(* Logix 5000 project; controller DC01 vendor 1 type 14 code 165 rev 32.12; software revision 32.04; part 3 of 13 *)
(* tags used below, declared in another part *)
   Break_1stStation : BOOL;
   Break_LineWide : BOOL;
   Break_WorkCenter : BOOL;
   Break_Workstation : BOOL;
   FaultExists : CONTROL;
   LN01_MainLine_MSG : MESSAGE;
   Local_Timer : TIMER[30];
   local_timer2 : TIMER;
   ONS_0 : DINT;
   Shift_Reset_ONS : BOOL;
   Barcode_Scan : MESSAGE;
   LN01_1st_Station_Break_Code : DINT;
   LN01_Boxing_MNT : DINT;
   LN01_Ceran_MNT : DINT;
   LN01_Console_MNT : DINT;
   LN01_Cooktop_MNT : DINT;
   LN01_Current_Shift_Duration_Mins : DINT;
   LN01_Current_Shift_Duration_wBreaks_Mins : DINT;
   LN01_DC_Controlled_Theoretical_Units : BOOL;
   LN01_Door_MNT : DINT;
   LN01_FPY : DINT;
   LN01_FrontFrame_MNT : DINT;
   LN01_Ignition_NewSNModel : BOOL[32];
   LN01_Ignition_SNModelMSG : STRING[5];
   LN01_MachineOverAll_MNT : DINT;
   LN01_Main_Messages : DINT[250];
   LN01_MainBack_MNT : DINT;
   LN01_Messages_Barcode_SNModel : Barcode_SNModel;
   LN01_OvenCavity_MNT : DINT;
   LN01_Schedule : UDT_Current_Status;
   LN01_Schedule_Cycle_Timer : TIMER;
   LN01_Schedule_Max_Break_Duration : DINT;
   LN01_Schedule_Max_Break_Timer : TIMER;
   LN01_Schedule_TAKT : REAL;
   LN01_Scheduled_Units_Buffer : DINT;
   LN01_SidePanels_MNT : DINT;
   LN01_StorageDrawer_MNT : DINT;
   LN01_Test_MNT : DINT;
   LN01_Theoretical_Units_Counter : COUNTER;
   LN01_Theoretical_Units_Counter_ONS : BOOL;
   LN01_Units_for_repair : DINT;
   LN01_Wiring_MNT : DINT;
   LN01ECM02 : DINT;
   LN01ECM03 : DINT;
   LN01ECM04 : DINT;
   LN01ECM05 : DINT;
   LN01EDM04 : DINT;
   LN01EDM06 : DINT;
   LN01EDM07 : DINT;
   LN01EDM08 : DINT;
   LN01EEM01 : DINT;
   LN01EEM02 : DINT;
   LN01EEM03 : DINT;
   LN01EES01 : DINT;
   LN01EES02 : DINT;
   LN01EES03 : DINT;
   LN01EES04 : DINT;
   LN01EFS04 : DINT;
   LN01EFS05 : DINT;
   LN01EGM04 : DINT;
   LN01EHM01 : DINT;
   LN01EHM02 : DINT;
   LN01EHM03 : DINT;
   LN01EHM04 : DINT;
   LN01EHM05 : DINT;
   LN01EHM06 : DINT;
   LN01EHM07 : DINT;
   LN01EHM08 : DINT;
   LN01NAS01 : DINT;
   LN01NAS02 : DINT;
   LN01NAS03 : DINT;
   LN01NBS02 : DINT;
   LN01SAS03 : DINT;
   LN01SBS01 : DINT;
   LN01SBS03 : DINT;
   LN01SFS03 : DINT;
   LN01WAM01 : DINT;
   LN01WBM01 : DINT;
   LN01WBM02 : DINT;
   LN01WBM03 : DINT;
   LN01WBM04 : DINT;
   LN01WCM01 : DINT;
   LN01WCM02 : DINT;
   LN01WCM03 : DINT;
   LN01WCM04 : DINT;
   LN01WCM05 : DINT;
   LN01WCM06 : DINT;
   LN01WDM01 : DINT;
   LN01WDM02 : DINT;
   LN01WDM03 : DINT;
   LN01WDM04 : DINT;
   LN01WDM05 : DINT;
   LN01WFS01 : DINT;
   LN01WFS02 : DINT;
   LN01WGM01 : DINT;
   LN01WGM02 : DINT;
   LN01WGM03 : DINT;
   LN01WGM04 : DINT;
   LN01WGM05 : DINT;
   LN01WHM08 : DINT;
(* LN01, continued *)

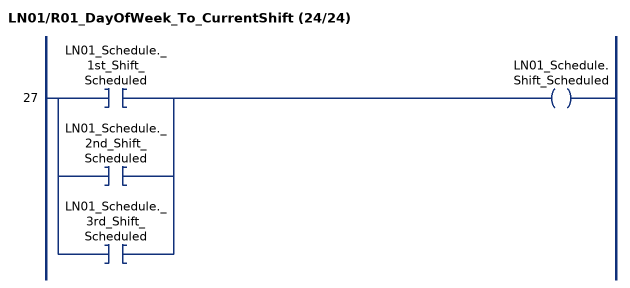
   [picture p24: LN01/R01_DayOfWeek_To_CurrentShift rungs 27-27]
   27: [XIC(LN01_Schedule._1st_Shift_Scheduled) ,XIC(LN01_Schedule._2nd_Shift_Scheduled) ,XIC(LN01_Schedule._3rd_Shift_Scheduled) ]OTE(LN01_Schedule.Shift_Scheduled);
END_ROUTINE

ROUTINE R02_CurrentShift_Calcs   (* ladder *)
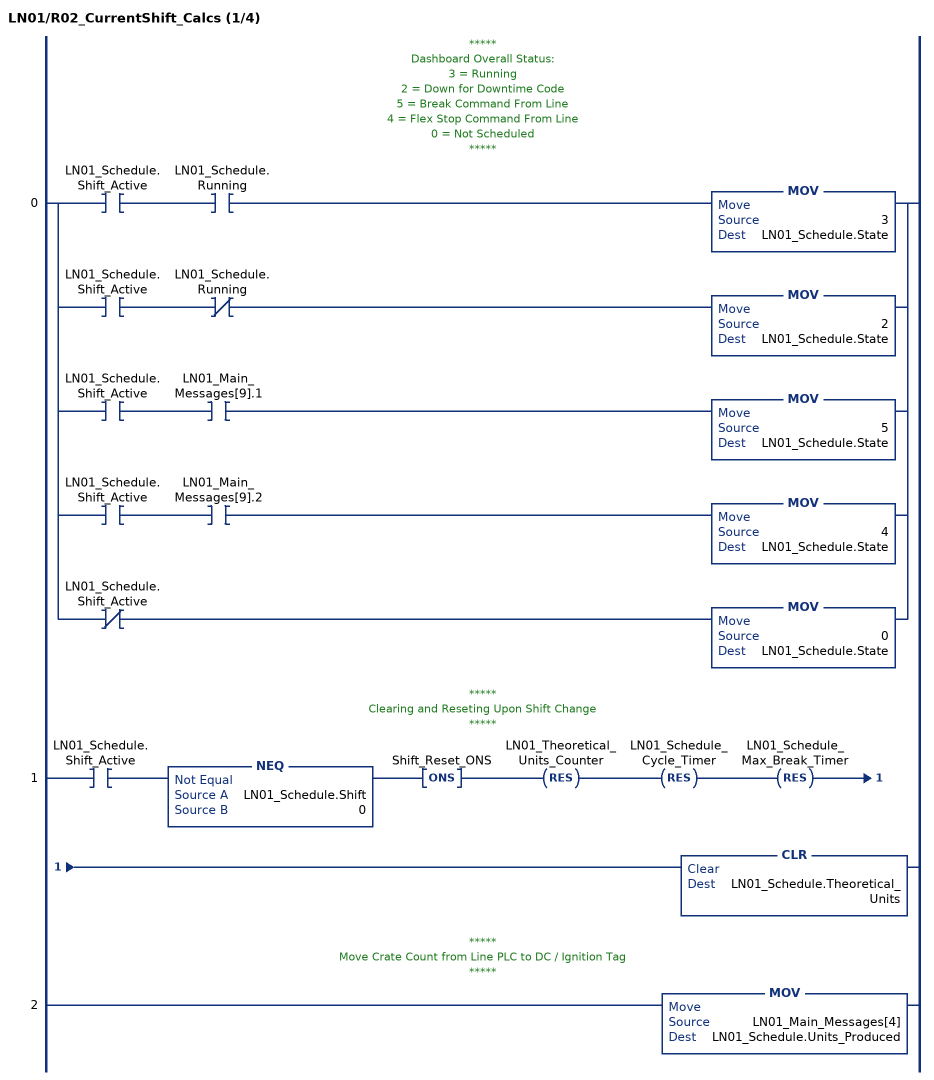
   // *****
   // Dashboard Overall Status:
   // 3 = Running
   // 2 = Down for Downtime Code
   // 5 = Break Command From Line
   // 4 = Flex Stop Command From Line
   // 0 = Not Scheduled
   // *****
   0: [XIC(LN01_Schedule.Shift_Active) XIC(LN01_Schedule.Running) MOV(3,LN01_Schedule.State) ,XIC(LN01_Schedule.Shift_Active) XIO(LN01_Schedule.Running) MOV(2,LN01_Schedule.State) ,XIC(LN01_Schedule.Shift_Active) XIC(LN01_Main_Messages[9].1) MOV(5,LN01_Schedule.State) ,XIC(LN01_Schedule.Shift_Active) XIC(LN01_Main_Messages[9].2) MOV(4,LN01_Schedule.State) ,XIO(LN01_Schedule.Shift_Active) MOV(0,LN01_Schedule.State) ];
   // *****
   // Clearing and Reseting Upon Shift Change
   // *****
   1: XIC(LN01_Schedule.Shift_Active)NEQ(LN01_Schedule.Shift,0)ONS(Shift_Reset_ONS)RES(LN01_Theoretical_Units_Counter)RES(LN01_Schedule_Cycle_Timer)RES(LN01_Schedule_Max_Break_Timer)CLR(LN01_Schedule.Theoretical_Units);
   // *****
   // Move Crate Count from Line PLC to DC / Ignition Tag
   // *****
   2: MOV(LN01_Main_Messages[4],LN01_Schedule.Units_Produced);
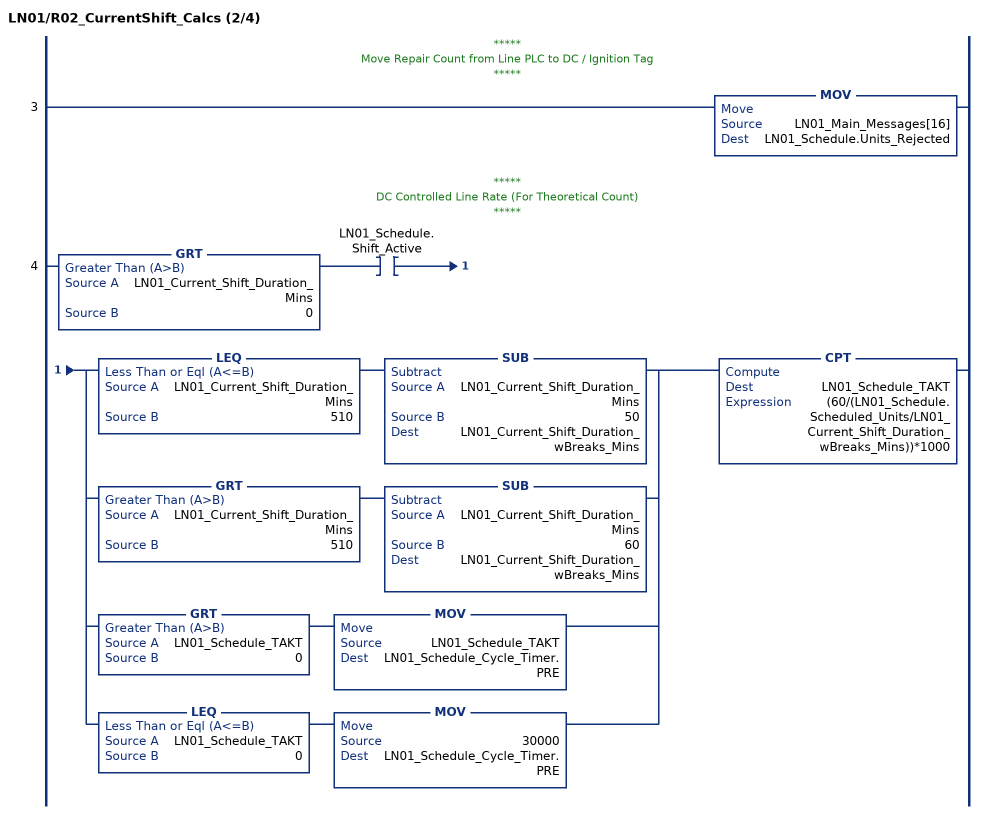
   // *****
   // Move Repair Count from Line PLC to DC / Ignition Tag
   // *****
   3: MOV(LN01_Main_Messages[16],LN01_Schedule.Units_Rejected);
   // *****
   // DC Controlled Line Rate (For Theoretical Count)
   // *****
   4: GRT(LN01_Current_Shift_Duration_Mins,0)XIC(LN01_Schedule.Shift_Active)[LEQ(LN01_Current_Shift_Duration_Mins,510) SUB(LN01_Current_Shift_Duration_Mins,50,LN01_Current_Shift_Duration_wBreaks_Mins) ,GRT(LN01_Current_Shift_Duration_Mins,510) SUB(LN01_Current_Shift_Duration_Mins,60,LN01_Current_Shift_Duration_wBreaks_Mins) ,GRT(LN01_Schedule_TAKT,0) MOV(LN01_Schedule_TAKT,LN01_Schedule_Cycle_Timer.PRE) ,LEQ(LN01_Schedule_TAKT,0) MOV(30000,LN01_Schedule_Cycle_Timer.PRE) ]CPT(LN01_Schedule_TAKT,(60/(LN01_Schedule.Scheduled_Units/LN01_Current_Shift_Duration_wBreaks_Mins))*1000);
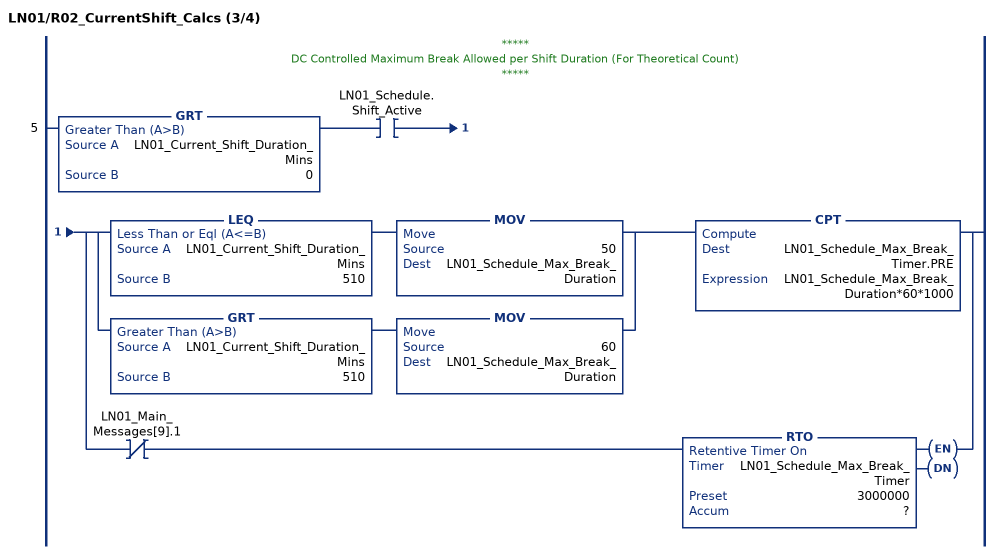
   // *****
   // DC Controlled Maximum Break Allowed per Shift Duration (For Theoretical Count)
   // *****
   5: GRT(LN01_Current_Shift_Duration_Mins,0)XIC(LN01_Schedule.Shift_Active)[[LEQ(LN01_Current_Shift_Duration_Mins,510) MOV(50,LN01_Schedule_Max_Break_Duration) ,GRT(LN01_Current_Shift_Duration_Mins,510) MOV(60,LN01_Schedule_Max_Break_Duration) ] CPT(LN01_Schedule_Max_Break_Timer.PRE,LN01_Schedule_Max_Break_Duration*60*1000) ,XIO(LN01_Main_Messages[9].1) RTO(LN01_Schedule_Max_Break_Timer,?,?) ];
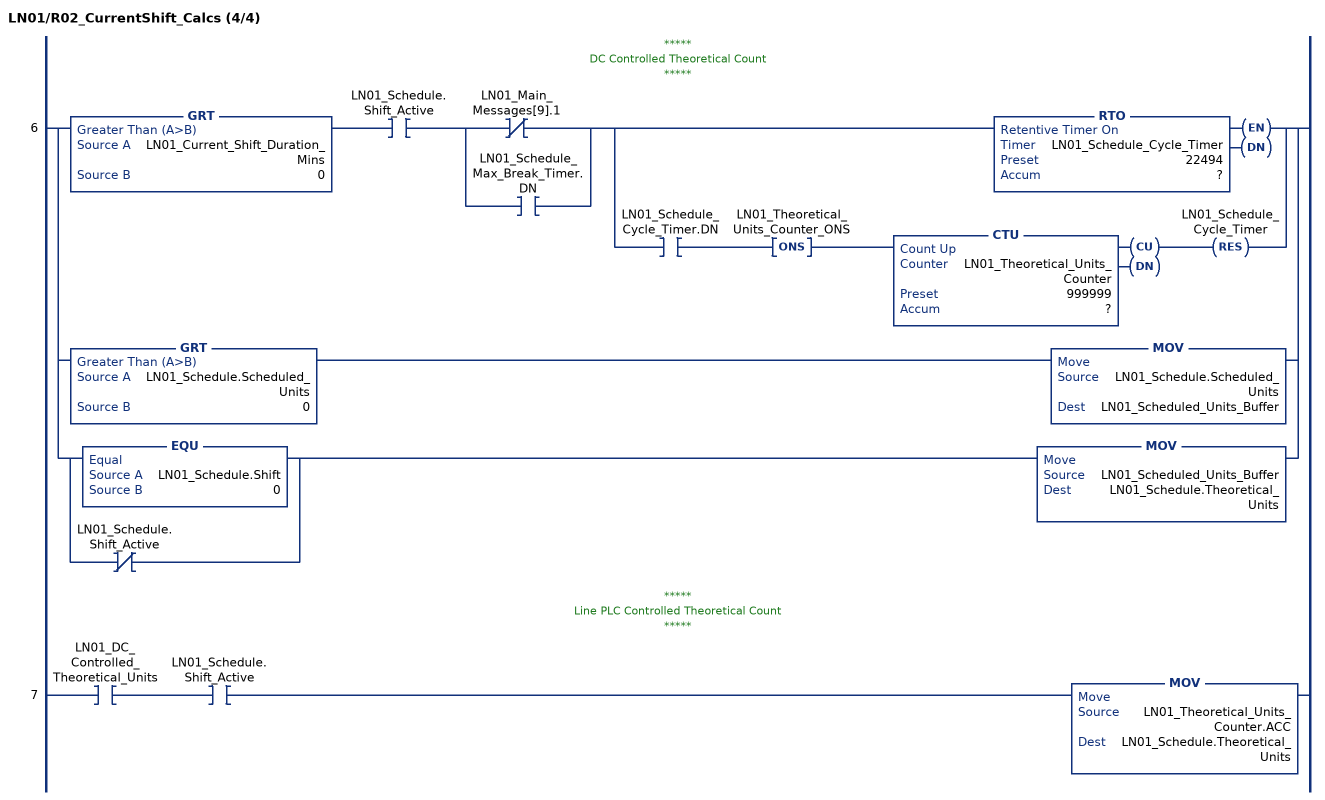
   // *****
   // DC Controlled Theoretical Count
   // *****
   6: [GRT(LN01_Current_Shift_Duration_Mins,0) XIC(LN01_Schedule.Shift_Active) [XIO(LN01_Main_Messages[9].1) ,XIC(LN01_Schedule_Max_Break_Timer.DN) ] [RTO(LN01_Schedule_Cycle_Timer,?,?) ,XIC(LN01_Schedule_Cycle_Timer.DN) ONS(LN01_Theoretical_Units_Counter_ONS) CTU(LN01_Theoretical_Units_Counter,?,?) RES(LN01_Schedule_Cycle_Timer) ] ,GRT(LN01_Schedule.Scheduled_Units,0) MOV(LN01_Schedule.Scheduled_Units,LN01_Scheduled_Units_Buffer) ,[EQU(LN01_Schedule.Shift,0) ,XIO(LN01_Schedule.Shift_Active) ] MOV(LN01_Scheduled_Units_Buffer,LN01_Schedule.Theoretical_Units) ];
   // *****
   // Line PLC Controlled Theoretical Count
   // *****
   7: XIC(LN01_DC_Controlled_Theoretical_Units)XIC(LN01_Schedule.Shift_Active)MOV(LN01_Theoretical_Units_Counter.ACC,LN01_Schedule.Theoretical_Units);
END_ROUTINE

ROUTINE R03_DataFromLines   (* ladder *)
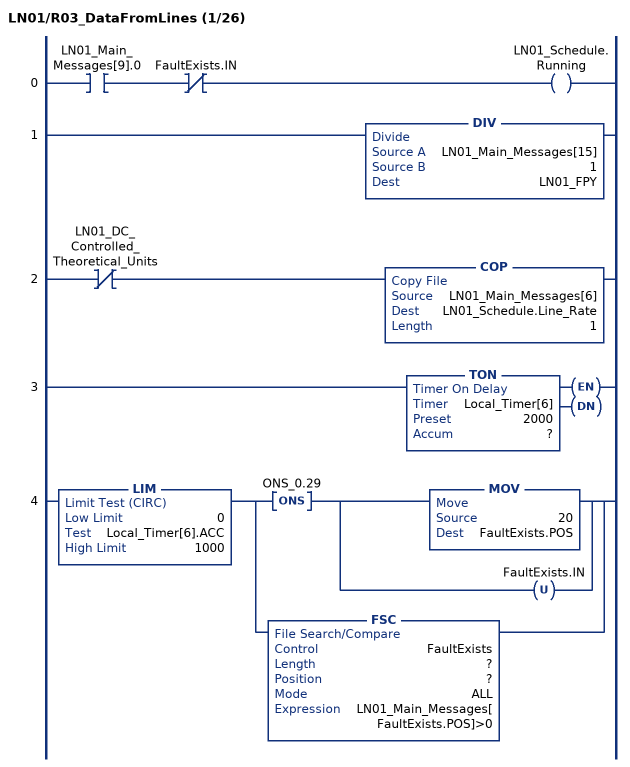
   0: XIC(LN01_Main_Messages[9].0)XIO(FaultExists.IN)OTE(LN01_Schedule.Running);
   1: DIV(LN01_Main_Messages[15],1,LN01_FPY);
   2: XIO(LN01_DC_Controlled_Theoretical_Units)COP(LN01_Main_Messages[6],LN01_Schedule.Line_Rate,1);
   3: TON(Local_Timer[6],?,?);
   4: LIM(0,Local_Timer[6].ACC,1000)[ONS(ONS_0.29) [MOV(20,FaultExists.POS) ,OTU(FaultExists.IN) ] ,FSC(FaultExists,?,?,ALL,LN01_Main_Messages[FaultExists.POS]>0) ];
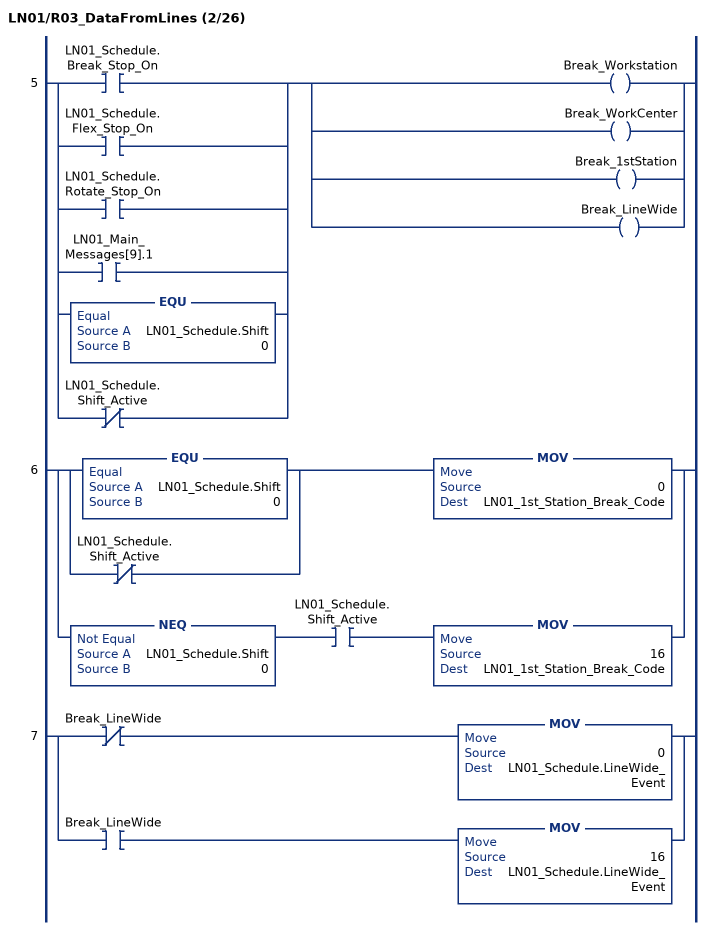
   5: [XIC(LN01_Schedule.Break_Stop_On) ,XIC(LN01_Schedule.Flex_Stop_On) ,XIC(LN01_Schedule.Rotate_Stop_On) ,XIC(LN01_Main_Messages[9].1) ,EQU(LN01_Schedule.Shift,0) ,XIO(LN01_Schedule.Shift_Active) ][OTE(Break_Workstation) ,OTE(Break_WorkCenter) ,OTE(Break_1stStation) ,OTE(Break_LineWide) ];
   6: [[EQU(LN01_Schedule.Shift,0) ,XIO(LN01_Schedule.Shift_Active) ] MOV(0,LN01_1st_Station_Break_Code) ,NEQ(LN01_Schedule.Shift,0) XIC(LN01_Schedule.Shift_Active) MOV(16,LN01_1st_Station_Break_Code) ];
   7: [XIO(Break_LineWide) MOV(0,LN01_Schedule.LineWide_Event) ,XIC(Break_LineWide) MOV(16,LN01_Schedule.LineWide_Event) ];
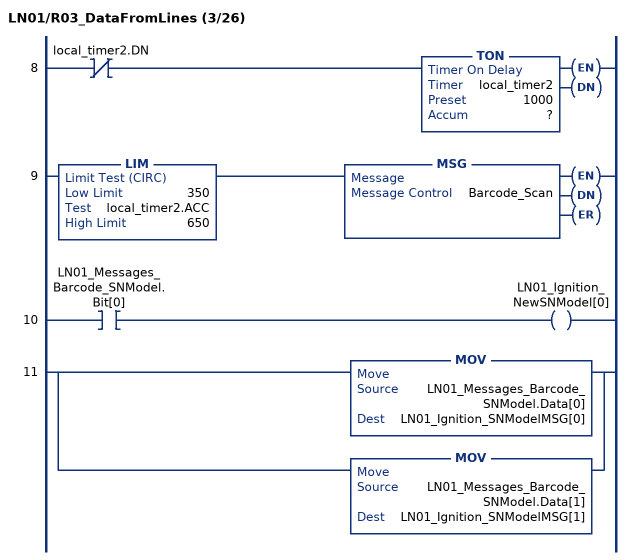
   8: XIO(local_timer2.DN)TON(local_timer2,?,?);
   9: LIM(350,local_timer2.ACC,650)MSG(Barcode_Scan);
   10: XIC(LN01_Messages_Barcode_SNModel.Bit[0])OTE(LN01_Ignition_NewSNModel[0]);
   11: [MOV(LN01_Messages_Barcode_SNModel.Data[0],LN01_Ignition_SNModelMSG[0]) ,MOV(LN01_Messages_Barcode_SNModel.Data[1],LN01_Ignition_SNModelMSG[1]) ];
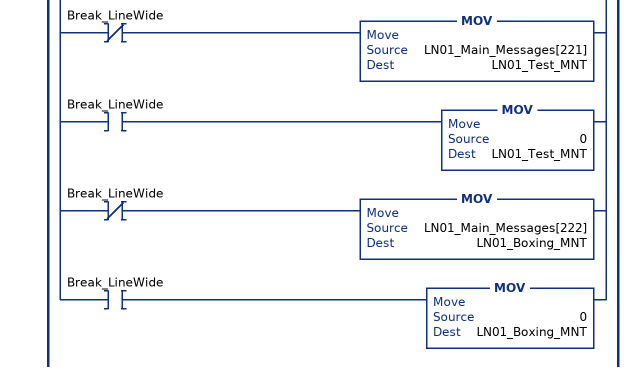
   // MNT Faults
   // If an MNT workcenter is tied to the main line or subline where there is already a workcenter with a workstaiton where "Break_LineWide (when high) MOVEs a 16 in, then that MNT can MOVE a 0 in when "Break_LineWide" goes high
   // If it is an independent MNT (not tied to a workcenter), "Break_LineWide" Tag should MOVE a 16 when "Break_LineWide" goes high
   12: [XIO(Break_LineWide) MOV(LN01_Main_Messages[20],LN01_MachineOverAll_MNT) ,XIC(Break_LineWide) MOV(0,LN01_MachineOverAll_MNT) ,XIO(Break_LineWide) MOV(LN01_Main_Messages[21],LN01_FrontFrame_MNT) ,XIC(Break_LineWide) MOV(0,LN01_FrontFrame_MNT) ,XIO(Break_LineWide) MOV(LN01_Main_Messages[22],LN01_OvenCavity_MNT) ,XIC(Break_LineWide) MOV(0,LN01_OvenCavity_MNT) ,XIO(Break_LineWide) MOV(LN01_Main_Messages[23],LN01_MainBack_MNT) ,XIC(Break_LineWide) MOV(0,LN01_MainBack_MNT) ,XIO(Break_LineWide) MOV(LN01_Main_Messages[24],LN01_SidePanels_MNT) ,XIC(Break_LineWide) MOV(0,LN01_SidePanels_MNT) ,XIO(Break_LineWide) MOV(LN01_Main_Messages[25],LN01_Console_MNT) ,XIC(Break_LineWide) MOV(0,LN01_Console_MNT) ,XIO(Break_LineWide) MOV(LN01_Main_Messages[26],LN01_Ceran_MNT) ,XIC(Break_LineWide) MOV(0,LN01_Ceran_MNT) ,XIO(Break_LineWide) MOV(LN01_Main_Messages[27],LN01_Cooktop_MNT) ,XIC(Break_LineWide) MOV(0,LN01_Cooktop_MNT) ,XIO(Break_LineWide) MOV(LN01_Main_Messages[28],LN01_Wiring_MNT) ,XIC(Break_LineWide) MOV(0,LN01_Wiring_MNT) ,XIO(Break_LineWide) MOV(LN01_Main_Messages[29],LN01_StorageDrawer_MNT) ,XIC(Break_LineWide) MOV(0,LN01_StorageDrawer_MNT) ,XIO(Break_LineWide) MOV(LN01_Main_Messages[220],LN01_Door_MNT) ,XIC(Break_LineWide) MOV(0,LN01_Door_MNT) ,XIO(Break_LineWide) MOV(LN01_Main_Messages[221],LN01_Test_MNT) ,XIC(Break_LineWide) MOV(0,LN01_Test_MNT) ,XIO(Break_LineWide) MOV(LN01_Main_Messages[222],LN01_Boxing_MNT) ,XIC(Break_LineWide) MOV(0,LN01_Boxing_MNT) ];
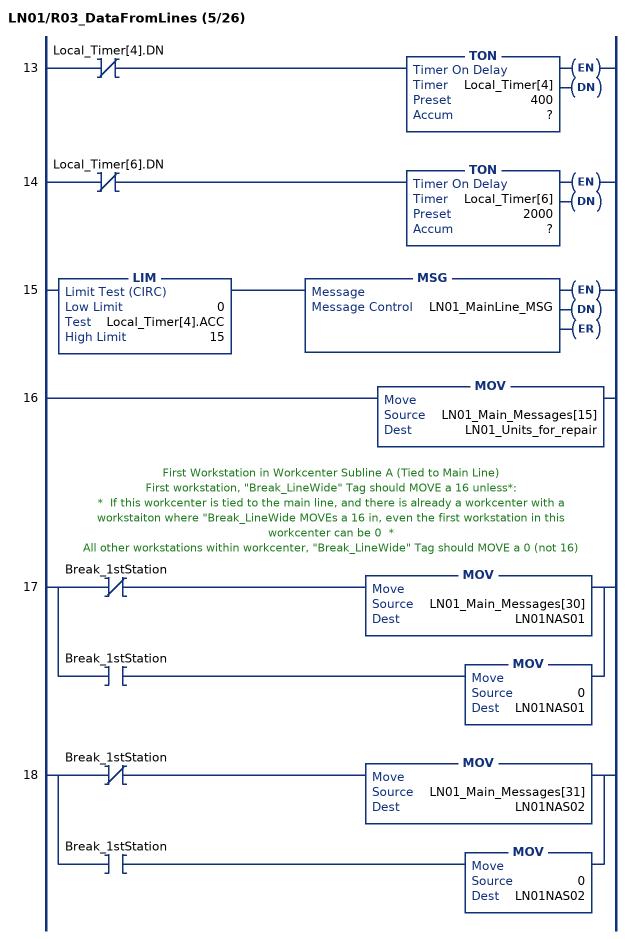
   13: XIO(Local_Timer[4].DN)TON(Local_Timer[4],?,?);
   14: XIO(Local_Timer[6].DN)TON(Local_Timer[6],?,?);
   15: LIM(0,Local_Timer[4].ACC,15)MSG(LN01_MainLine_MSG);
   16: MOV(LN01_Main_Messages[15],LN01_Units_for_repair);
   // First Workstation in Workcenter Subline A (Tied to Main Line)
   // First workstation, "Break_LineWide" Tag should MOVE a 16 unless*:
   // *  If this workcenter is tied to the main line, and there is already a workcenter with a workstaiton where "Break_LineWide MOVEs a 16 in, even the first workstation in this workcenter can be 0  *
   // All other workstations within workcenter, "Break_LineWide" Tag should MOVE a 0 (not 16)
   17: [XIO(Break_1stStation) MOV(LN01_Main_Messages[30],LN01NAS01) ,XIC(Break_1stStation) MOV(0,LN01NAS01) ];
   18: [XIO(Break_1stStation) MOV(LN01_Main_Messages[31],LN01NAS02) ,XIC(Break_1stStation) MOV(0,LN01NAS02) ];
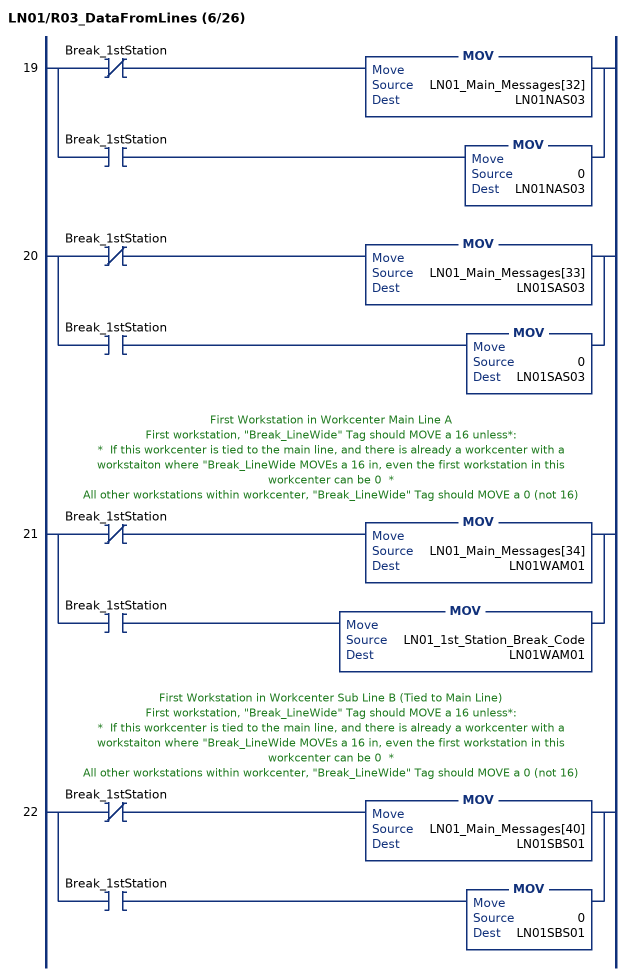
   19: [XIO(Break_1stStation) MOV(LN01_Main_Messages[32],LN01NAS03) ,XIC(Break_1stStation) MOV(0,LN01NAS03) ];
   20: [XIO(Break_1stStation) MOV(LN01_Main_Messages[33],LN01SAS03) ,XIC(Break_1stStation) MOV(0,LN01SAS03) ];
   // First Workstation in Workcenter Main Line A
   // First workstation, "Break_LineWide" Tag should MOVE a 16 unless*:
   // *  If this workcenter is tied to the main line, and there is already a workcenter with a workstaiton where "Break_LineWide MOVEs a 16 in, even the first workstation in this workcenter can be 0  *
   // All other workstations within workcenter, "Break_LineWide" Tag should MOVE a 0 (not 16)
   21: [XIO(Break_1stStation) MOV(LN01_Main_Messages[34],LN01WAM01) ,XIC(Break_1stStation) MOV(LN01_1st_Station_Break_Code,LN01WAM01) ];
   // First Workstation in Workcenter Sub Line B (Tied to Main Line)
   // First workstation, "Break_LineWide" Tag should MOVE a 16 unless*:
   // *  If this workcenter is tied to the main line, and there is already a workcenter with a workstaiton where "Break_LineWide MOVEs a 16 in, even the first workstation in this workcenter can be 0  *
   // All other workstations within workcenter, "Break_LineWide" Tag should MOVE a 0 (not 16)
   22: [XIO(Break_1stStation) MOV(LN01_Main_Messages[40],LN01SBS01) ,XIC(Break_1stStation) MOV(0,LN01SBS01) ];
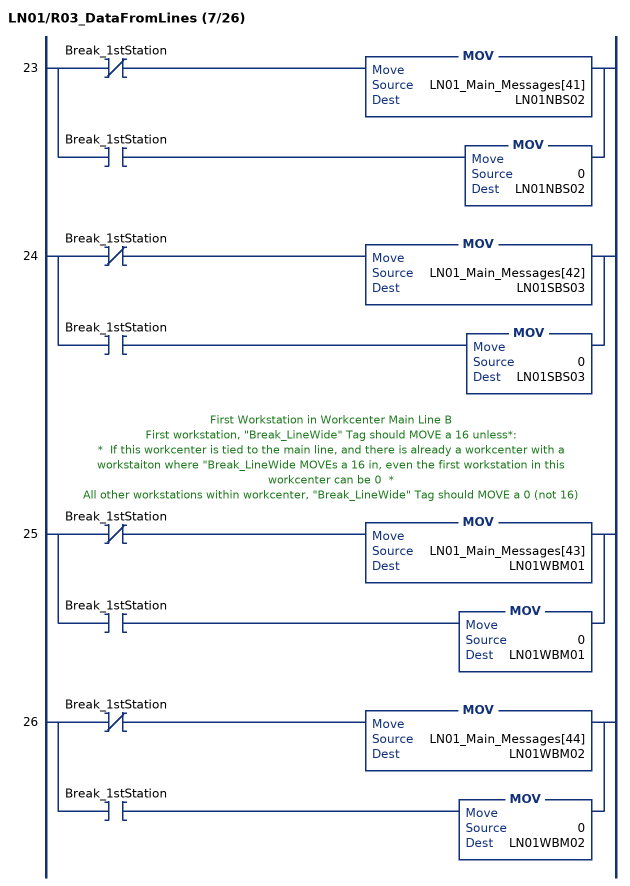
   23: [XIO(Break_1stStation) MOV(LN01_Main_Messages[41],LN01NBS02) ,XIC(Break_1stStation) MOV(0,LN01NBS02) ];
   24: [XIO(Break_1stStation) MOV(LN01_Main_Messages[42],LN01SBS03) ,XIC(Break_1stStation) MOV(0,LN01SBS03) ];
   // First Workstation in Workcenter Main Line B
   // First workstation, "Break_LineWide" Tag should MOVE a 16 unless*:
   // *  If this workcenter is tied to the main line, and there is already a workcenter with a workstaiton where "Break_LineWide MOVEs a 16 in, even the first workstation in this workcenter can be 0  *
   // All other workstations within workcenter, "Break_LineWide" Tag should MOVE a 0 (not 16)
   25: [XIO(Break_1stStation) MOV(LN01_Main_Messages[43],LN01WBM01) ,XIC(Break_1stStation) MOV(0,LN01WBM01) ];
   26: [XIO(Break_1stStation) MOV(LN01_Main_Messages[44],LN01WBM02) ,XIC(Break_1stStation) MOV(0,LN01WBM02) ];
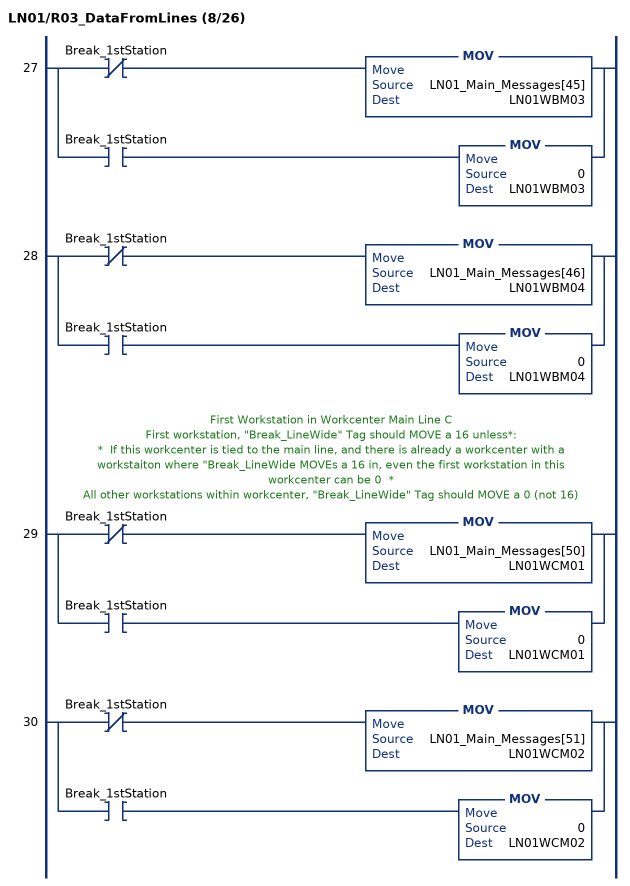
   27: [XIO(Break_1stStation) MOV(LN01_Main_Messages[45],LN01WBM03) ,XIC(Break_1stStation) MOV(0,LN01WBM03) ];
   28: [XIO(Break_1stStation) MOV(LN01_Main_Messages[46],LN01WBM04) ,XIC(Break_1stStation) MOV(0,LN01WBM04) ];
   // First Workstation in Workcenter Main Line C
   // First workstation, "Break_LineWide" Tag should MOVE a 16 unless*:
   // *  If this workcenter is tied to the main line, and there is already a workcenter with a workstaiton where "Break_LineWide MOVEs a 16 in, even the first workstation in this workcenter can be 0  *
   // All other workstations within workcenter, "Break_LineWide" Tag should MOVE a 0 (not 16)
   29: [XIO(Break_1stStation) MOV(LN01_Main_Messages[50],LN01WCM01) ,XIC(Break_1stStation) MOV(0,LN01WCM01) ];
   30: [XIO(Break_1stStation) MOV(LN01_Main_Messages[51],LN01WCM02) ,XIC(Break_1stStation) MOV(0,LN01WCM02) ];
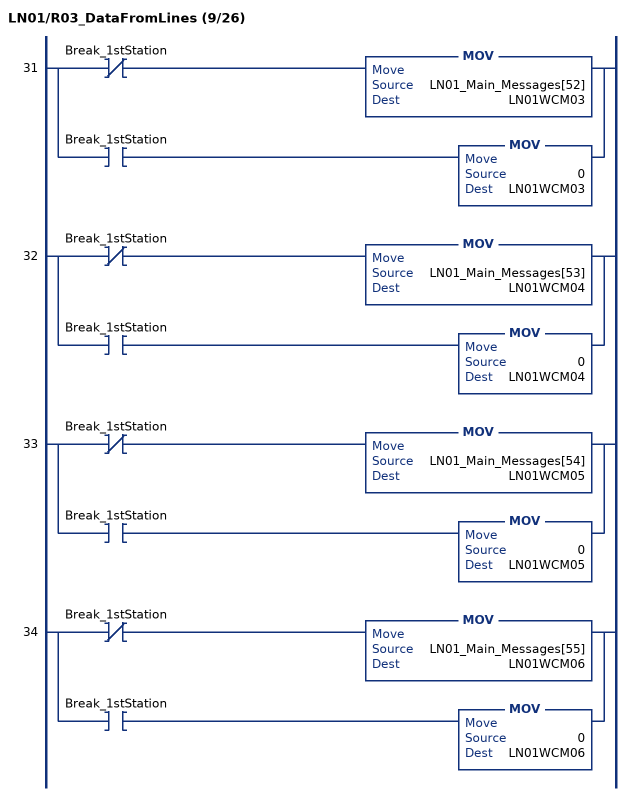
   31: [XIO(Break_1stStation) MOV(LN01_Main_Messages[52],LN01WCM03) ,XIC(Break_1stStation) MOV(0,LN01WCM03) ];
   32: [XIO(Break_1stStation) MOV(LN01_Main_Messages[53],LN01WCM04) ,XIC(Break_1stStation) MOV(0,LN01WCM04) ];
   33: [XIO(Break_1stStation) MOV(LN01_Main_Messages[54],LN01WCM05) ,XIC(Break_1stStation) MOV(0,LN01WCM05) ];
   34: [XIO(Break_1stStation) MOV(LN01_Main_Messages[55],LN01WCM06) ,XIC(Break_1stStation) MOV(0,LN01WCM06) ];
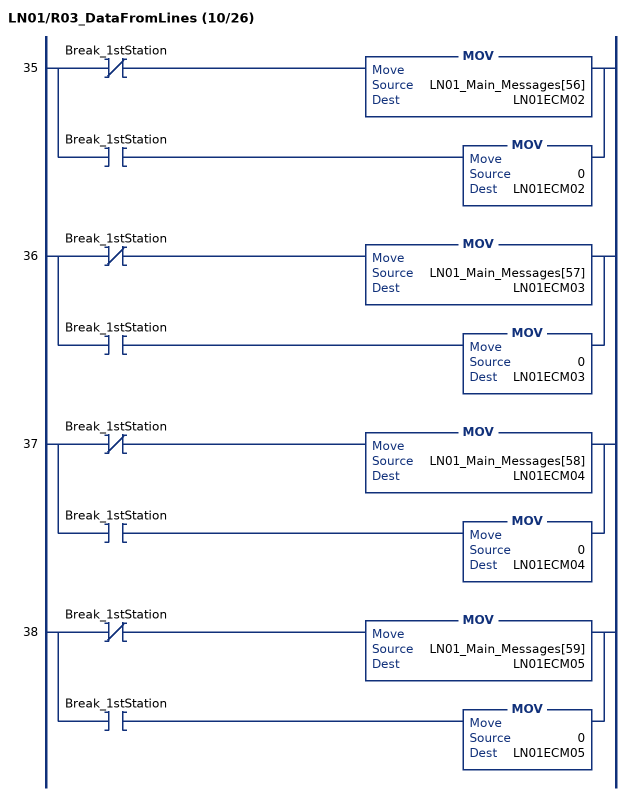
   35: [XIO(Break_1stStation) MOV(LN01_Main_Messages[56],LN01ECM02) ,XIC(Break_1stStation) MOV(0,LN01ECM02) ];
   36: [XIO(Break_1stStation) MOV(LN01_Main_Messages[57],LN01ECM03) ,XIC(Break_1stStation) MOV(0,LN01ECM03) ];
   37: [XIO(Break_1stStation) MOV(LN01_Main_Messages[58],LN01ECM04) ,XIC(Break_1stStation) MOV(0,LN01ECM04) ];
   38: [XIO(Break_1stStation) MOV(LN01_Main_Messages[59],LN01ECM05) ,XIC(Break_1stStation) MOV(0,LN01ECM05) ];
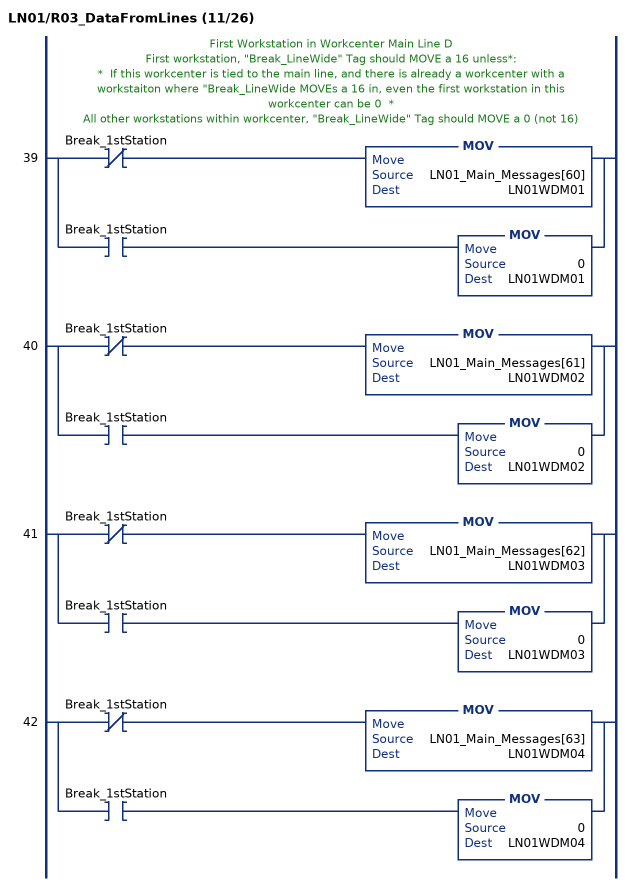
   // First Workstation in Workcenter Main Line D
   // First workstation, "Break_LineWide" Tag should MOVE a 16 unless*:
   // *  If this workcenter is tied to the main line, and there is already a workcenter with a workstaiton where "Break_LineWide MOVEs a 16 in, even the first workstation in this workcenter can be 0  *
   // All other workstations within workcenter, "Break_LineWide" Tag should MOVE a 0 (not 16)
   39: [XIO(Break_1stStation) MOV(LN01_Main_Messages[60],LN01WDM01) ,XIC(Break_1stStation) MOV(0,LN01WDM01) ];
   40: [XIO(Break_1stStation) MOV(LN01_Main_Messages[61],LN01WDM02) ,XIC(Break_1stStation) MOV(0,LN01WDM02) ];
   41: [XIO(Break_1stStation) MOV(LN01_Main_Messages[62],LN01WDM03) ,XIC(Break_1stStation) MOV(0,LN01WDM03) ];
   42: [XIO(Break_1stStation) MOV(LN01_Main_Messages[63],LN01WDM04) ,XIC(Break_1stStation) MOV(0,LN01WDM04) ];
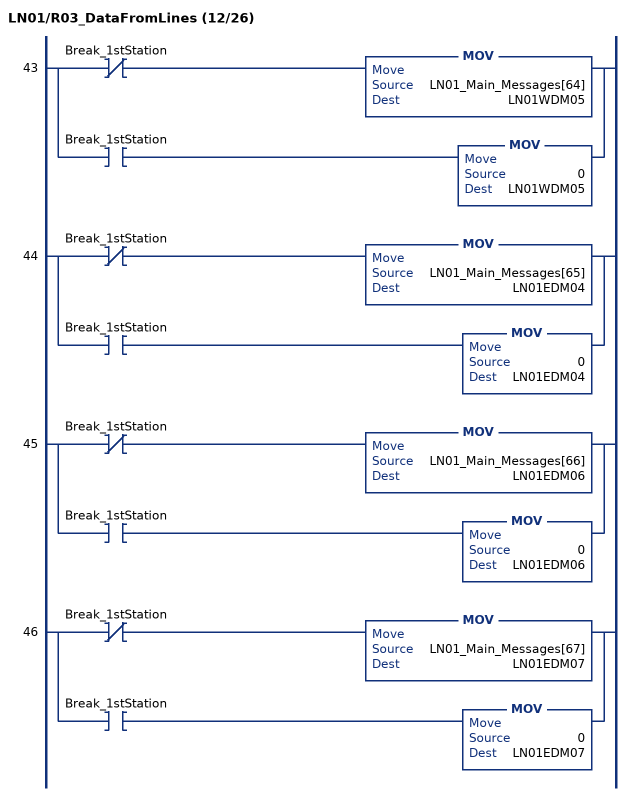
   43: [XIO(Break_1stStation) MOV(LN01_Main_Messages[64],LN01WDM05) ,XIC(Break_1stStation) MOV(0,LN01WDM05) ];
   44: [XIO(Break_1stStation) MOV(LN01_Main_Messages[65],LN01EDM04) ,XIC(Break_1stStation) MOV(0,LN01EDM04) ];
   45: [XIO(Break_1stStation) MOV(LN01_Main_Messages[66],LN01EDM06) ,XIC(Break_1stStation) MOV(0,LN01EDM06) ];
   46: [XIO(Break_1stStation) MOV(LN01_Main_Messages[67],LN01EDM07) ,XIC(Break_1stStation) MOV(0,LN01EDM07) ];
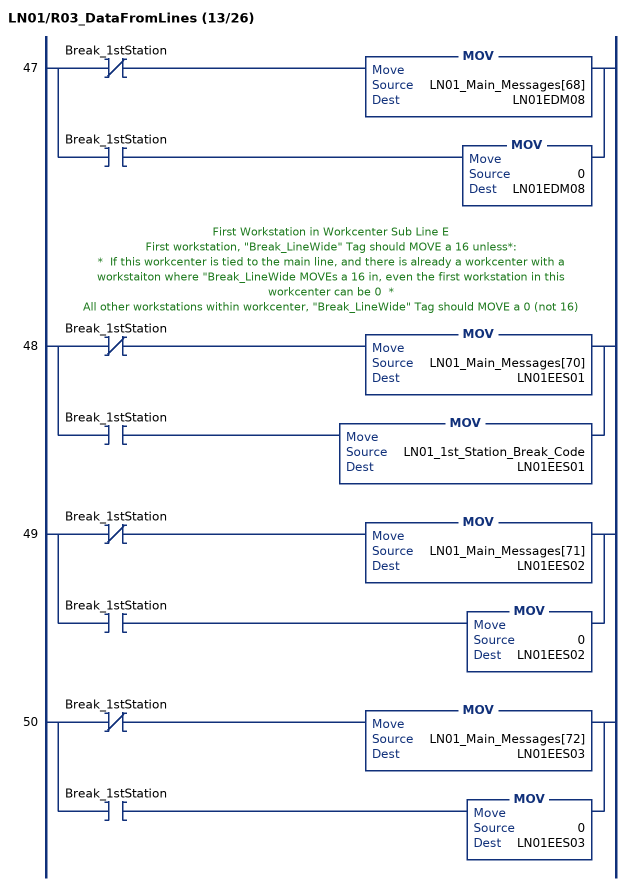
   47: [XIO(Break_1stStation) MOV(LN01_Main_Messages[68],LN01EDM08) ,XIC(Break_1stStation) MOV(0,LN01EDM08) ];
   // First Workstation in Workcenter Sub Line E
   // First workstation, "Break_LineWide" Tag should MOVE a 16 unless*:
   // *  If this workcenter is tied to the main line, and there is already a workcenter with a workstaiton where "Break_LineWide MOVEs a 16 in, even the first workstation in this workcenter can be 0  *
   // All other workstations within workcenter, "Break_LineWide" Tag should MOVE a 0 (not 16)
   48: [XIO(Break_1stStation) MOV(LN01_Main_Messages[70],LN01EES01) ,XIC(Break_1stStation) MOV(LN01_1st_Station_Break_Code,LN01EES01) ];
   49: [XIO(Break_1stStation) MOV(LN01_Main_Messages[71],LN01EES02) ,XIC(Break_1stStation) MOV(0,LN01EES02) ];
   50: [XIO(Break_1stStation) MOV(LN01_Main_Messages[72],LN01EES03) ,XIC(Break_1stStation) MOV(0,LN01EES03) ];
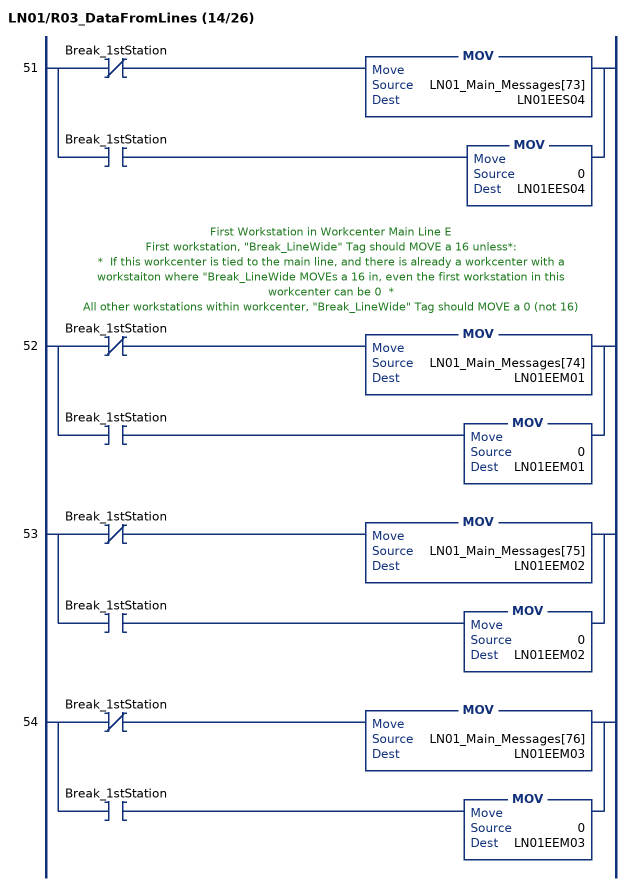
   51: [XIO(Break_1stStation) MOV(LN01_Main_Messages[73],LN01EES04) ,XIC(Break_1stStation) MOV(0,LN01EES04) ];
   // First Workstation in Workcenter Main Line E
   // First workstation, "Break_LineWide" Tag should MOVE a 16 unless*:
   // *  If this workcenter is tied to the main line, and there is already a workcenter with a workstaiton where "Break_LineWide MOVEs a 16 in, even the first workstation in this workcenter can be 0  *
   // All other workstations within workcenter, "Break_LineWide" Tag should MOVE a 0 (not 16)
   52: [XIO(Break_1stStation) MOV(LN01_Main_Messages[74],LN01EEM01) ,XIC(Break_1stStation) MOV(0,LN01EEM01) ];
   53: [XIO(Break_1stStation) MOV(LN01_Main_Messages[75],LN01EEM02) ,XIC(Break_1stStation) MOV(0,LN01EEM02) ];
   54: [XIO(Break_1stStation) MOV(LN01_Main_Messages[76],LN01EEM03) ,XIC(Break_1stStation) MOV(0,LN01EEM03) ];
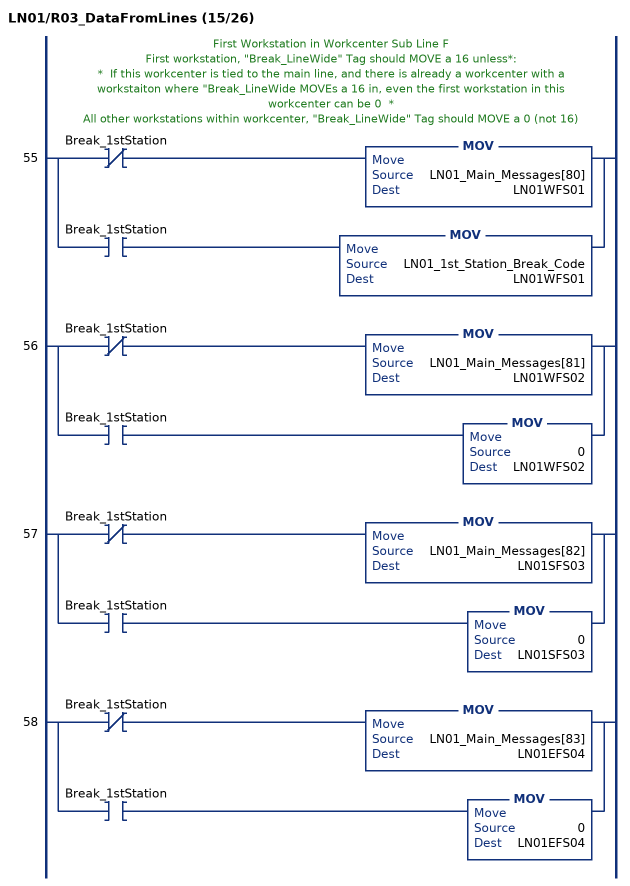
   // First Workstation in Workcenter Sub Line F
   // First workstation, "Break_LineWide" Tag should MOVE a 16 unless*:
   // *  If this workcenter is tied to the main line, and there is already a workcenter with a workstaiton where "Break_LineWide MOVEs a 16 in, even the first workstation in this workcenter can be 0  *
   // All other workstations within workcenter, "Break_LineWide" Tag should MOVE a 0 (not 16)
   55: [XIO(Break_1stStation) MOV(LN01_Main_Messages[80],LN01WFS01) ,XIC(Break_1stStation) MOV(LN01_1st_Station_Break_Code,LN01WFS01) ];
   56: [XIO(Break_1stStation) MOV(LN01_Main_Messages[81],LN01WFS02) ,XIC(Break_1stStation) MOV(0,LN01WFS02) ];
   57: [XIO(Break_1stStation) MOV(LN01_Main_Messages[82],LN01SFS03) ,XIC(Break_1stStation) MOV(0,LN01SFS03) ];
   58: [XIO(Break_1stStation) MOV(LN01_Main_Messages[83],LN01EFS04) ,XIC(Break_1stStation) MOV(0,LN01EFS04) ];
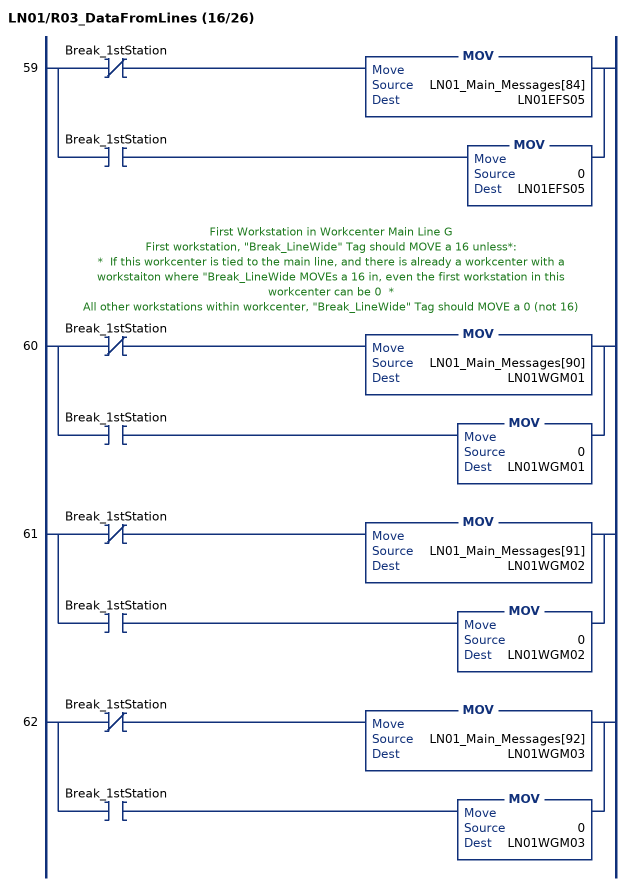
   59: [XIO(Break_1stStation) MOV(LN01_Main_Messages[84],LN01EFS05) ,XIC(Break_1stStation) MOV(0,LN01EFS05) ];
   // First Workstation in Workcenter Main Line G
   // First workstation, "Break_LineWide" Tag should MOVE a 16 unless*:
   // *  If this workcenter is tied to the main line, and there is already a workcenter with a workstaiton where "Break_LineWide MOVEs a 16 in, even the first workstation in this workcenter can be 0  *
   // All other workstations within workcenter, "Break_LineWide" Tag should MOVE a 0 (not 16)
   60: [XIO(Break_1stStation) MOV(LN01_Main_Messages[90],LN01WGM01) ,XIC(Break_1stStation) MOV(0,LN01WGM01) ];
   61: [XIO(Break_1stStation) MOV(LN01_Main_Messages[91],LN01WGM02) ,XIC(Break_1stStation) MOV(0,LN01WGM02) ];
   62: [XIO(Break_1stStation) MOV(LN01_Main_Messages[92],LN01WGM03) ,XIC(Break_1stStation) MOV(0,LN01WGM03) ];
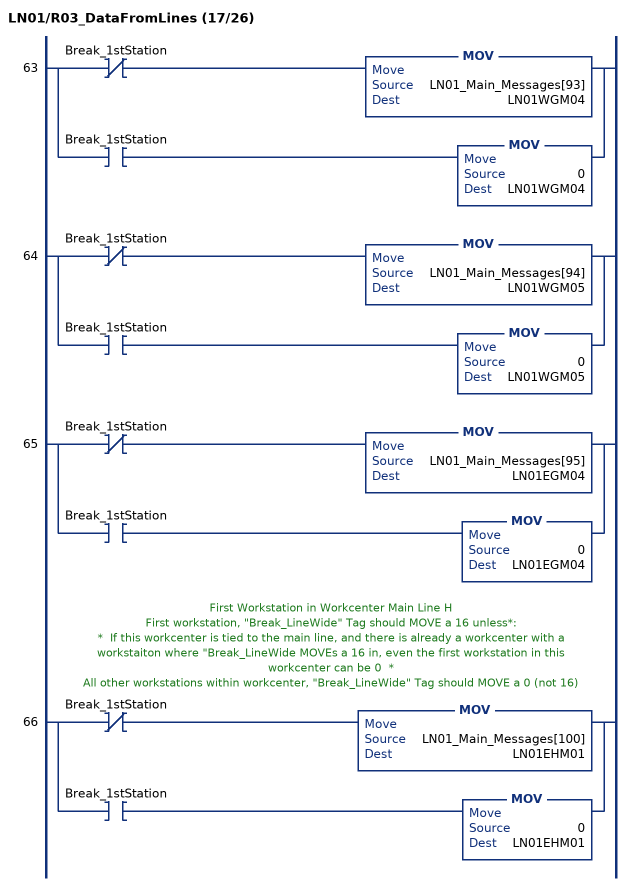
   63: [XIO(Break_1stStation) MOV(LN01_Main_Messages[93],LN01WGM04) ,XIC(Break_1stStation) MOV(0,LN01WGM04) ];
   64: [XIO(Break_1stStation) MOV(LN01_Main_Messages[94],LN01WGM05) ,XIC(Break_1stStation) MOV(0,LN01WGM05) ];
   65: [XIO(Break_1stStation) MOV(LN01_Main_Messages[95],LN01EGM04) ,XIC(Break_1stStation) MOV(0,LN01EGM04) ];
   // First Workstation in Workcenter Main Line H
   // First workstation, "Break_LineWide" Tag should MOVE a 16 unless*:
   // *  If this workcenter is tied to the main line, and there is already a workcenter with a workstaiton where "Break_LineWide MOVEs a 16 in, even the first workstation in this workcenter can be 0  *
   // All other workstations within workcenter, "Break_LineWide" Tag should MOVE a 0 (not 16)
   66: [XIO(Break_1stStation) MOV(LN01_Main_Messages[100],LN01EHM01) ,XIC(Break_1stStation) MOV(0,LN01EHM01) ];
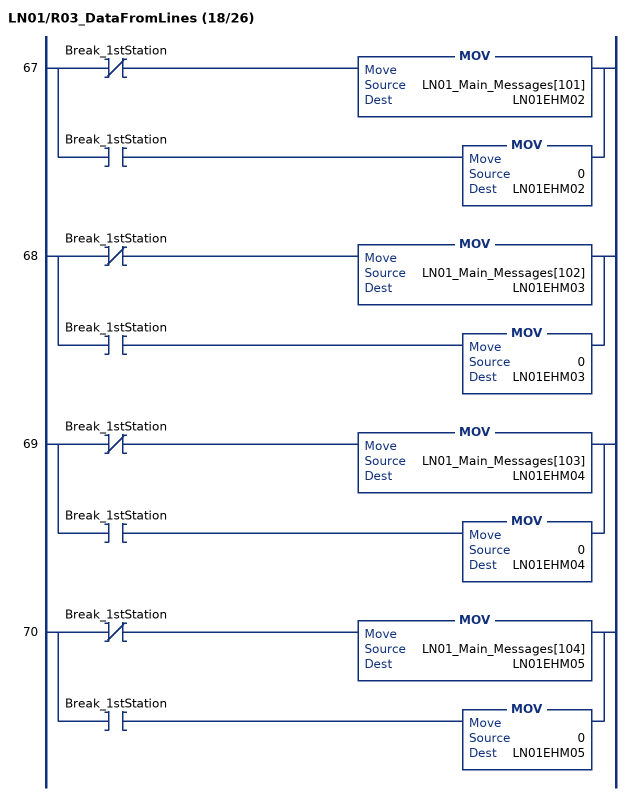
   67: [XIO(Break_1stStation) MOV(LN01_Main_Messages[101],LN01EHM02) ,XIC(Break_1stStation) MOV(0,LN01EHM02) ];
   68: [XIO(Break_1stStation) MOV(LN01_Main_Messages[102],LN01EHM03) ,XIC(Break_1stStation) MOV(0,LN01EHM03) ];
   69: [XIO(Break_1stStation) MOV(LN01_Main_Messages[103],LN01EHM04) ,XIC(Break_1stStation) MOV(0,LN01EHM04) ];
   70: [XIO(Break_1stStation) MOV(LN01_Main_Messages[104],LN01EHM05) ,XIC(Break_1stStation) MOV(0,LN01EHM05) ];
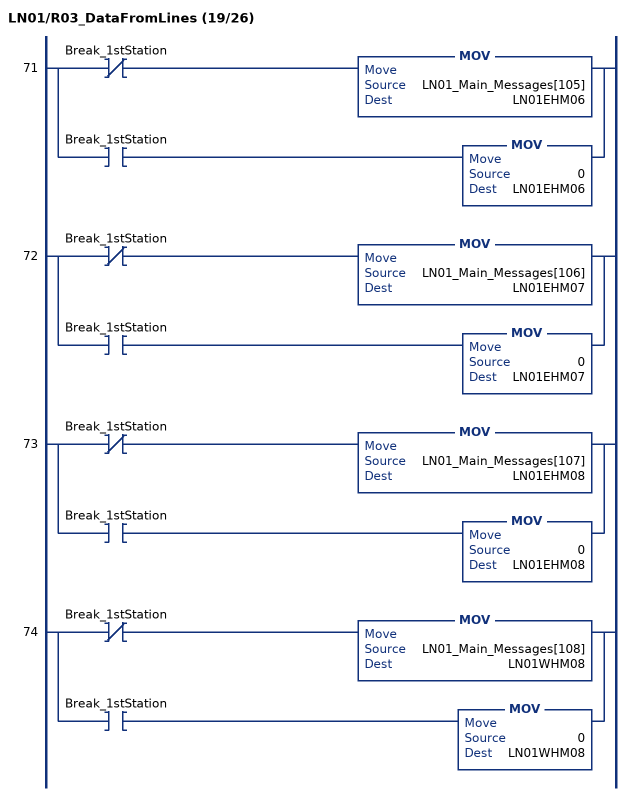
   71: [XIO(Break_1stStation) MOV(LN01_Main_Messages[105],LN01EHM06) ,XIC(Break_1stStation) MOV(0,LN01EHM06) ];
   72: [XIO(Break_1stStation) MOV(LN01_Main_Messages[106],LN01EHM07) ,XIC(Break_1stStation) MOV(0,LN01EHM07) ];
   73: [XIO(Break_1stStation) MOV(LN01_Main_Messages[107],LN01EHM08) ,XIC(Break_1stStation) MOV(0,LN01EHM08) ];
   74: [XIO(Break_1stStation) MOV(LN01_Main_Messages[108],LN01WHM08) ,XIC(Break_1stStation) MOV(0,LN01WHM08) ];
